# EPICS autosave request: vici/fourGasSelect_positions.req
$(P)$(Q):SELECT.FRST
$(P)$(Q):SELECT.FVST
$(P)$(Q):SELECT.ONST
$(P)$(Q):SELECT.SVST
$(P)$(Q):SELECT.SXST
$(P)$(Q):SELECT.THST
$(P)$(Q):SELECT.TWST
$(P)$(Q):SELECT.ZRST
